FUNCTION_BLOCK AngularAcceleration EXTENDS SM_AngularAcceleration
VAR_INPUT
END_VAR
VAR_OUTPUT
END_VAR
VAR
    _testVar : INT;
END_VAR

SUPER^();

END_FUNCTION_BLOCK

(* stored: Version 1.1.0.1, ProductVersion 3.1.4018.5
   POU AngularAcceleration: Id {0b51a99b-520f-4d3f-bd6d-77d631952085}, SpecialFunc None *)
